FUNCTION_BLOCK Discrete_PI_REAL2 (* Composite Function Block Type *)
  (* Standard: 61499-2 *)
  (* Version 0.0, 2018-07-31, 4DIAC-IDE, 4DIAC-Consortium *)
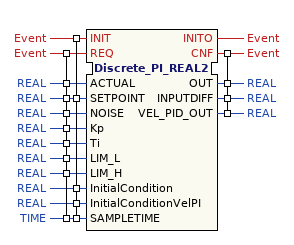
  EVENT_INPUT
    INIT WITH SAMPLETIME, SETPOINT, InitialCondition, InitialConditionVelPI; (* Initialization Request *)
    REQ WITH SAMPLETIME, ACTUAL, SETPOINT, NOISE, Kp, Ti, LIM_L, LIM_H; (* Normal Execution Request *)
  END_EVENT
  EVENT_OUTPUT
    INITO; (* Initialization Confirm *)
    CNF WITH OUT, INPUTDIFF, VEL_PID_OUT; (* Execution Confirmation *)
  END_EVENT
  VAR_INPUT
    ACTUAL : REAL;
    SETPOINT : REAL;
    NOISE : REAL;
    Kp : REAL;
    Ti : REAL;
    LIM_L : REAL;
    LIM_H : REAL;
    InitialCondition : REAL;
    InitialConditionVelPI : REAL;
    SAMPLETIME : TIME;
  END_VAR
  VAR_OUTPUT
    OUT : REAL;
    INPUTDIFF : REAL;
    VEL_PID_OUT : REAL;
  END_VAR
  FBS
    F_ADD : F_ADD;
    F_FT_LIMIT : F_FT_LIMIT;
    Velocity_PI_REAL2 : Velocity_PI_REAL2;
    Delay_With_InitConditionREALtype : Delay_With_InitConditionREALtype;
  END_FBS
  EVENT_CONNECTIONS
    INIT TO Velocity_PI_REAL2.INIT;
    REQ TO Velocity_PI_REAL2.REQ;
    REQ TO F_FT_LIMIT.REQ;
    Velocity_PI_REAL2.INITO TO INITO;
    Velocity_PI_REAL2.CNF TO F_ADD.REQ;
    Velocity_PI_REAL2.CNF TO CNF;
    Velocity_PI_REAL2.INITO TO Delay_With_InitConditionREALtype.INIT;
    REQ TO Delay_With_InitConditionREALtype.Start_and_REQ;
    F_FT_LIMIT.CNF TO Delay_With_InitConditionREALtype.Start_and_REQ;
    Delay_With_InitConditionREALtype.CNF TO F_ADD.REQ;
    Delay_With_InitConditionREALtype.CNF TO CNF;
    F_ADD.CNF TO F_FT_LIMIT.REQ;
  END_CONNECTIONS
  DATA_CONNECTIONS
    ACTUAL TO Velocity_PI_REAL2.ACTUAL;
    SETPOINT TO Velocity_PI_REAL2.SETPOINT;
    NOISE TO Velocity_PI_REAL2.NOISE;
    Kp TO Velocity_PI_REAL2.Kp;
    Ti TO Velocity_PI_REAL2.Ti;
    InitialConditionVelPI TO Velocity_PI_REAL2.InitialCondition;
    SAMPLETIME TO Velocity_PI_REAL2.SAMPLETIME_ECYCLE;
    LIM_L TO F_FT_LIMIT.LIM_L;
    LIM_H TO F_FT_LIMIT.LIM_H;
    Velocity_PI_REAL2.DELTAOUTPUT TO F_ADD.IN1;
    Velocity_PI_REAL2.DELTAOUTPUT TO VEL_PID_OUT;
    Velocity_PI_REAL2.INPUTDIFF TO INPUTDIFF;
    F_FT_LIMIT.OUT TO Delay_With_InitConditionREALtype.DelayedInput;
    Delay_With_InitConditionREALtype.OUT TO F_ADD.IN2;
    Delay_With_InitConditionREALtype.OUT TO OUT;
    InitialCondition TO Delay_With_InitConditionREALtype.InitialCondition;
    SAMPLETIME TO Delay_With_InitConditionREALtype.DelayTime;
    F_ADD.OUT TO F_FT_LIMIT.VAL;
  END_CONNECTIONS
END_FUNCTION_BLOCK
